// TwinCAT 3 PLC project PLC1
// ProgramVersion: 3.1.4023.0
// libraries:
//   Tc2_BA, * (Beckhoff Automation GmbH)
//   Tc2_Standard, * (Beckhoff Automation GmbH)
//   Tc2_System, * (Beckhoff Automation GmbH)
//   Tc3_Module, * (Beckhoff Automation GmbH)
// project tree:
//   GVLs/ GVL_Fill.TcGVL
//   / PlcTask.TcTTO
//   POUs/ Conveyor.TcPOU, MAIN.TcPOU, Pump.TcPOU, Seal.TcPOU
// real-time tasks:
//   TASK PlcTask: cycle T#10ms, priority 20, ADS port 350

CONFIGURATION PLC1
    RESOURCE PLC ON TwinCAT3
        TASK PlcTask(INTERVAL := T#10ms, PRIORITY := 20);
        PROGRAM MAIN WITH PlcTask : MAIN;
    END_RESOURCE
END_CONFIGURATION

// ---- GVLs/GVL_Fill.TcGVL
{attribute 'qualified_only'}
VAR_GLOBAL
	bStart AT %I* : BOOL := FALSE;
	mStart AT %Q* : BOOL;
	bStop AT %I* : BOOL := FALSE;
	bEmergency : BOOL := FALSE;
	fbBA: FB_BA_PIDCtrl;
END_VAR

// ---- POUs/MAIN.TcPOU
PROGRAM MAIN
VAR
	Activate : BOOL;
	bLed : BOOL := FALSE;
	Timer1 : BOOL := FALSE;
	Timer2 : BOOL := FALSE;
	fbT2 : TON;
	fbT3 : TON;
	Init: BOOL := TRUE;
END_VAR

Pump();
Seal();
Conveyor();
IF Init AND GVL_Fill.bStart THEN
	fbT2(IN := FALSE);
	fbT3(IN := FALSE);
	Init := FALSE;
END_IF
IF NOT GVL_Fill.bEmergency THEN
	IF NOT GVL_Fill.bStop THEN
		IF GVL_Fill.bStart THEN
			Activate := TRUE;
		END_IF
		IF Activate THEN
			GVL_Fill.mStart := TRUE;
			bLed := TRUE;
		ELSE
			GVL_Fill.mStart := FALSE;
			bLed := FALSE;
		END_IF
	ELSE
		fbT3(IN := TRUE, PT := T#1S, Q => Timer2);
		IF Timer2 THEN
			fbT3(IN := FALSE);
			GVL_Fill.bStop := FALSE;
			Timer2 := FALSE;
		END_IF
		//GVL_Fill.bStop := FALSE;
		Activate := FALSE;
		bLed := FALSE;
		Init := TRUE;
	END_IF
ELSE
	GVL_Fill.bStop := FALSE;
	GVL_Fill.bStart := FALSE;
	GVL_Fill.mStart := FALSE;
	Activate := FALSE;
	bLed := FALSE;
	Init := TRUE;
END_IF

END_PROGRAM

// ---- POUs/Pump.TcPOU
PROGRAM Pump
VAR_INPUT
	height : 	LREAL;
	diameter : 	LREAL := 2;
	volume :	LREAL := 25.13;
	fbT1 :		TON;
	FlowValve1 : LREAL := 0;
	FlowValve2 : LREAL := 0;
	FlowSensor1 : LREAL := 0;
	FlowSensor2 : LREAL := 0;
	bValve1Opened			: BOOL;
	bValve2Opened			: BOOL;
	Bottle :	LREAL := 0;
	countFill :	INT := 0;
	// tMove: TIME;
	ClockFill: BOOL := FALSE;
END_VAR
VAR
	ActValve : BOOL := TRUE;
	ActFill : BOOL := TRUE;
	Check_Fill: BOOL := FALSE;
	//ReadyMove1 : BOOL := FALSE;
	//ActMove1: BOOL := FALSE;
END_VAR

//Cylinder Tank: Diameter = 500, Height = 1000
FlowSensor1 := FlowValve1; FlowSensor2 := FlowValve2;
volume := volume + (FlowValve1 - FlowValve2)/100;
height := (4 * volume)/(pi * EXPT(diameter, 2));
IF MAIN.Activate THEN
	IF height >= 9 THEN //Upper level sensor
		FlowValve1 := 0;
		bValve1Opened := FALSE;
	END_IF
	IF height <= 8 THEN //Lower level sensor
		FlowValve1 := 0.251;
		bValve1Opened := TRUE;
	END_IF
	IF NOT ClockFill THEN 
		FlowValve2 := 0.25; 
		bValve2Opened := TRUE;
	ELSE 
		FlowValve2 := 0; 
		bValve2Opened := FALSE;
		JMP label1; //Jump to label1
	END_IF 
	IF countFill >= 1 THEN 
		Seal.enableSeal := TRUE; 
	END_IF
	IF FlowValve2 = 0.25 AND ActFill AND Conveyor.Pos_Bottle1 = 400 THEN
		Bottle := Bottle + FlowValve2/100;
		IF Bottle >= 0.5 AND NOT Check_Fill THEN
			ActFill := FALSE; // Stop Filling
			Check_Fill := TRUE; //Ensure ActFill interrupted once
		END_IF
		IF Bottle >= 0.5 AND Check_Fill THEN
			Bottle := 0;
			countFill := countFill + 1; // Counting Filled Bottle
			// Wait for Transmission
			label1 : fbT1(IN := Check_Fill, PT := T#1S, Q => ActFill);
			ClockFill := TRUE;
			IF ActFill THEN
				fbT1(IN := FALSE);
				Check_Fill := FALSE;
				ClockFill := FALSE;
			END_IF
		END_IF
	END_IF
END_IF

IF NOT MAIN.Activate THEN
	Bottle := 0; height := 8.95;
	FlowValve1 := 0; FlowValve2 := 0;
	countFill := 0; ActFill := TRUE; Check_Fill := FALSE;
	ClockFill := FALSE;
	IF GVL_Fill.bEmergency THEN
		ActValve := FALSE;
	END_IF
END_IF

END_PROGRAM

// ---- POUs/Seal.TcPOU
PROGRAM Seal
VAR_INPUT
	ActSeal : 		BOOL := TRUE;
	PosSeal : 		LREAL := 0;
	Rotate : 		INT := 0;
	t2 : 			INT := 0;
	t3 : 			INT := 0;
	t4 : 			INT := 0;
	Check_Rotate :	BOOL := FALSE;
	ClockSeal : 	BOOL := FALSE;
	countSeal :		INT := -10;
	G :				BOOL := FALSE;
	enableSeal :	BOOL := FALSE;
	bSealed				: BOOL;
END_VAR

IF MAIN.Activate THEN
	IF Pump.ClockFill THEN //Clock from Pump
		ActSeal := FALSE;
		JMP label2; 
	ELSE ActSeal := TRUE; 
	END_IF //Sealing process includes 3 steps (in 2 seconds)
	IF ActSeal AND Conveyor.Pos_Bottle2 = 800 AND enableSeal THEN
		t2 := t2 + 1; //Step 1: Capping machine moves down (in 0.4 second)
		IF t2 >= 40 THEN t2 := 40; END_IF
		PosSeal := 250 * t2/100;
		IF PosSeal = 100 THEN
			t4 := t4 + 1; //Step 2: The cowl rotates and tightens the cap (in 1.2 second)
			IF t4 >= 120 THEN t4 := 120; END_IF
			Rotate := t4;
			IF Rotate = 120 THEN Check_Rotate := TRUE; END_IF
			IF Check_Rotate THEN
				bSealed := TRUE;
				t3 := t3 + 1; //Step 3: Capping machine moves up (in 0.4 second)
				IF t3 >= 40 THEN t3 := 40; END_IF
				PosSeal := 100 - 250 * t3/100;
				IF ActSeal := FALSE THEN
					label2 : t2 := 0; t3 := 0; t4 := 0;
					countSeal := Pump.countFill - 1; G := TRUE;
					IF G THEN
						Check_Rotate := FALSE;
						Rotate := 0; PosSeal := 0; G := FALSE;
					END_IF
				END_IF
			END_IF
		END_IF
	END_IF
END_IF

IF NOT MAIN.Activate THEN
	ActSeal := TRUE; t2 := 0; t3 := 0; t4 := 0; PosSeal := 0; Rotate := 0;
	Check_Rotate := FALSE;
	ClockSeal := FALSE;
	countSeal := -10; G := FALSE;
	enableSeal := FALSE;
END_IF

END_PROGRAM

// ---- POUs/Conveyor.TcPOU
PROGRAM Conveyor
VAR_INPUT
	ActMotor 		: BOOL := FALSE;
	RunMotor 		: BOOL := FALSE;
	vMotor 			: LREAL := 400;
	fMotorSpeed		: LREAL;
	Pos_Bottle0 	: LREAL := 0; //Position Variable of Bottle 0
	Pos_Bottle1 	: LREAL := 400; //Position Variable of Bottle 1
	Pos_Bottle2 	: LREAL := 800; //Position Variable of Bottle 2
	j 				: INT := 0;
END_VAR

IF MAIN.Activate THEN
	ActMotor := TRUE;
	IF Pump.ClockFill THEN
		RunMotor := TRUE;
		fMotorSpeed := vMotor;
		j := j + 1;
		IF j >= 100 THEN j := 100; END_IF
		Pos_Bottle0 := 0 + vMotor * j/100; //Increasing by time
		Pos_Bottle1 := 400 + vMotor * j/100; 
		Pos_Bottle2 := 800 + vMotor * j/100; 
		IF j = 100 THEN //Equal 1 second of transmission
			Seal.bSealed := FALSE;
			Pos_Bottle0 := 0; // Reset the value
			Pos_Bottle1 := 400;
			Pos_Bottle2 := 800;
			j := 0;
		END_IF
	ELSE
		RunMotor := FALSE;
		fMotorSpeed := 0;
	END_IF
END_IF

IF NOT MAIN.Activate THEN
	ActMotor := FALSE;
	RunMotor := FALSE; j := 0;
	Pos_Bottle0 := 0;
	Pos_Bottle1 := 400;
	Pos_Bottle2 := 800;
END_IF

END_PROGRAM
